% RSLogix 500 project PV5.RSS, saved by version 8.30.00.16 %
PROJECT "PV5"    % processor: Bul.1763 MicroLogix 1100 Series B %

PROGRAM FILES
  LAD 2   25 rungs

DATA FILES
  O0 OUTPUT  5 elements
  I1 INPUT  7 elements
  S2 STATUS  66 elements
  B3 BINARY  2 elements
  T4 TIMER  3 elements
  C5 COUNTER  1 elements
  R6 CONTROL  1 elements
  N7 INTEGER  3 elements
  F8 FLOAT  1 elements

LADDER 2
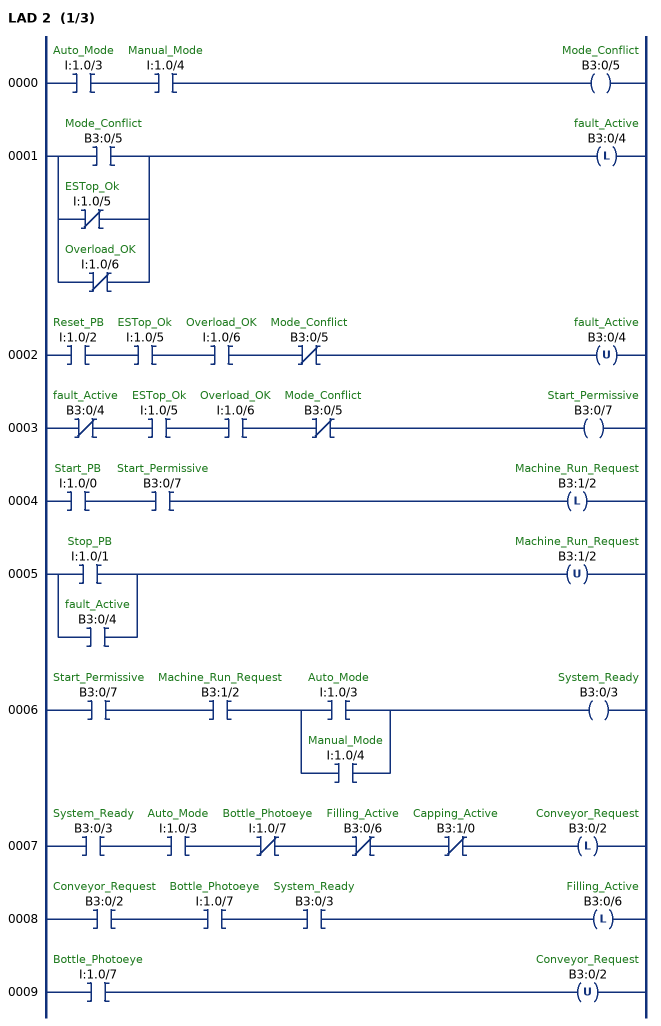
% Rung: 0 %
SOR XIC I:1.0/3 XIC I:1.0/4 OTE B3:0/5 EOR
%   I:1.0/3  "Auto_Mode" %
%   I:1.0/4  "Manual_Mode" %
%   B3:0/5  "Mode_Conflict" %
% Rung: 1 %
SOR BST XIC B3:0/5 NXB BST XIO I:1.0/5 NXB XIO I:1.0/6 BND BND OTL B3:0/4 EOR
%   B3:0/5  "Mode_Conflict" %
%   I:1.0/5  "ESTop_Ok" %
%   I:1.0/6  "Overload_OK" %
%   B3:0/4  "fault_Active" %
% Rung: 2 %
SOR XIC I:1.0/2 XIC I:1.0/5 XIC I:1.0/6 XIO B3:0/5 OTU B3:0/4 EOR
%   I:1.0/2  "Reset_PB" %
%   I:1.0/5  "ESTop_Ok" %
%   I:1.0/6  "Overload_OK" %
%   B3:0/5  "Mode_Conflict" %
%   B3:0/4  "fault_Active" %
% Rung: 3 %
SOR XIO B3:0/4 XIC I:1.0/5 XIC I:1.0/6 XIO B3:0/5 OTE B3:0/7 EOR
%   B3:0/4  "fault_Active" %
%   I:1.0/5  "ESTop_Ok" %
%   I:1.0/6  "Overload_OK" %
%   B3:0/5  "Mode_Conflict" %
%   B3:0/7  "Start_Permissive" %
% Rung: 4 %
SOR XIC I:1.0/0 XIC B3:0/7 OTL B3:1/2 EOR
%   I:1.0/0  "Start_PB" %
%   B3:0/7  "Start_Permissive" %
%   B3:1/2  "Machine_Run_Request" %
% Rung: 5 %
SOR BST XIC I:1.0/1 NXB XIC B3:0/4 BND OTU B3:1/2 EOR
%   I:1.0/1  "Stop_PB" %
%   B3:0/4  "fault_Active" %
%   B3:1/2  "Machine_Run_Request" %
% Rung: 6 %
SOR XIC B3:0/7 XIC B3:1/2 BST XIC I:1.0/3 NXB XIC I:1.0/4 BND OTE B3:0/3 EOR
%   B3:0/7  "Start_Permissive" %
%   B3:1/2  "Machine_Run_Request" %
%   I:1.0/3  "Auto_Mode" %
%   I:1.0/4  "Manual_Mode" %
%   B3:0/3  "System_Ready" %
% Rung: 7 %
SOR XIC B3:0/3 XIC I:1.0/3 XIO I:1.0/7 XIO B3:0/6 XIO B3:1/0 OTL B3:0/2 EOR
%   B3:0/3  "System_Ready" %
%   I:1.0/3  "Auto_Mode" %
%   I:1.0/7  "Bottle_Photoeye" %
%   B3:0/6  "Filling_Active" %
%   B3:1/0  "Capping_Active" %
%   B3:0/2  "Conveyor_Request" %
% Rung: 8 %
SOR XIC B3:0/2 XIC I:1.0/7 XIC B3:0/3 OTL B3:0/6 EOR
%   B3:0/2  "Conveyor_Request" %
%   I:1.0/7  "Bottle_Photoeye" %
%   B3:0/3  "System_Ready" %
%   B3:0/6  "Filling_Active" %
% Rung: 9 %
SOR XIC I:1.0/7 OTU B3:0/2 EOR
%   I:1.0/7  "Bottle_Photoeye" %
%   B3:0/2  "Conveyor_Request" %

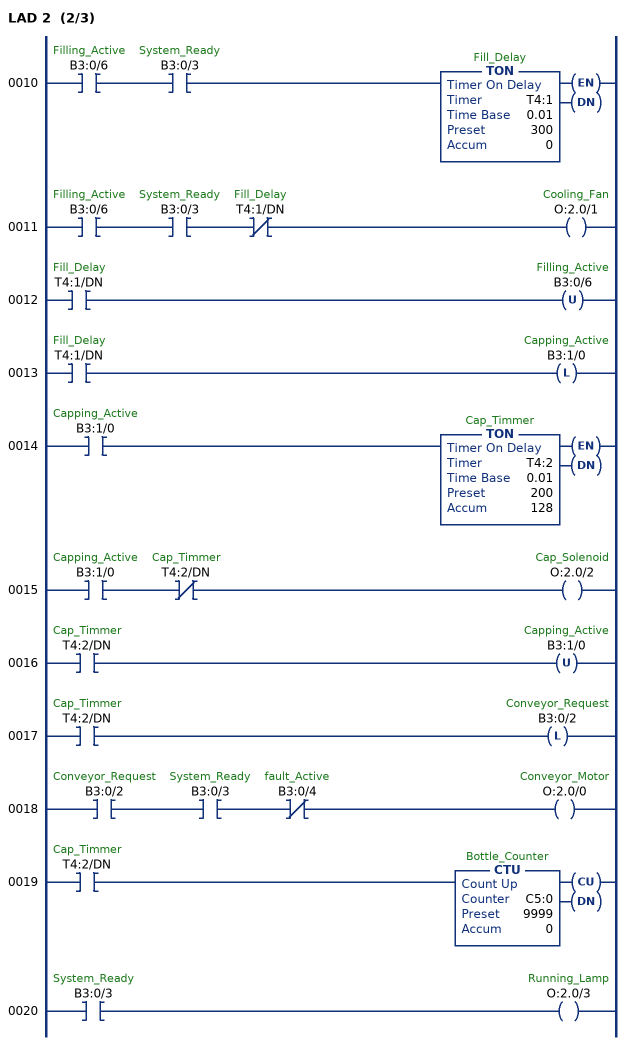
% Rung: 10 %
SOR XIC B3:0/6 XIC B3:0/3 TON T4:1 0.01 300 0 EOR
%   B3:0/6  "Filling_Active" %
%   B3:0/3  "System_Ready" %
%   T4:1  "Fill_Delay" %
% Rung: 11 %
SOR XIC B3:0/6 XIC B3:0/3 XIO T4:1/DN OTE O:2.0/1 EOR
%   B3:0/6  "Filling_Active" %
%   B3:0/3  "System_Ready" %
%   T4:1  "Fill_Delay" %
%   O:2.0/1  "Cooling_Fan" %
% Rung: 12 %
SOR XIC T4:1/DN OTU B3:0/6 EOR
%   T4:1  "Fill_Delay" %
%   B3:0/6  "Filling_Active" %
% Rung: 13 %
SOR XIC T4:1/DN OTL B3:1/0 EOR
%   T4:1  "Fill_Delay" %
%   B3:1/0  "Capping_Active" %
% Rung: 14 %
SOR XIC B3:1/0 TON T4:2 0.01 200 128 EOR
%   B3:1/0  "Capping_Active" %
%   T4:2  "Cap_Timmer" %
% Rung: 15 %
SOR XIC B3:1/0 XIO T4:2/DN OTE O:2.0/2 EOR
%   B3:1/0  "Capping_Active" %
%   T4:2  "Cap_Timmer" %
%   O:2.0/2  "Cap_Solenoid" %
% Rung: 16 %
SOR XIC T4:2/DN OTU B3:1/0 EOR
%   T4:2  "Cap_Timmer" %
%   B3:1/0  "Capping_Active" %
% Rung: 17 %
SOR XIC T4:2/DN OTL B3:0/2 EOR
%   T4:2  "Cap_Timmer" %
%   B3:0/2  "Conveyor_Request" %
% Rung: 18 %
SOR XIC B3:0/2 XIC B3:0/3 XIO B3:0/4 OTE O:2.0/0 EOR
%   B3:0/2  "Conveyor_Request" %
%   B3:0/3  "System_Ready" %
%   B3:0/4  "fault_Active" %
%   O:2.0/0  "Conveyor_Motor" %
% Rung: 19 %
SOR XIC T4:2/DN CTU C5:0 9999 0 EOR
%   T4:2  "Cap_Timmer" %
%   C5:0  "Bottle_Counter" %
% Rung: 20 %
SOR XIC B3:0/3 OTE O:2.0/3 EOR
%   B3:0/3  "System_Ready" %
%   O:2.0/3  "Running_Lamp" %

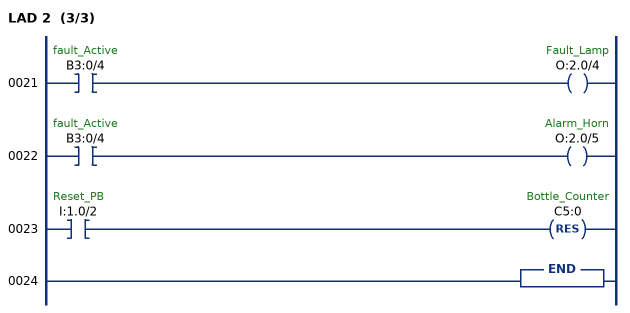
% Rung: 21 %
SOR XIC B3:0/4 OTE O:2.0/4 EOR
%   B3:0/4  "fault_Active" %
%   O:2.0/4  "Fault_Lamp" %
% Rung: 22 %
SOR XIC B3:0/4 OTE O:2.0/5 EOR
%   B3:0/4  "fault_Active" %
%   O:2.0/5  "Alarm_Horn" %
% Rung: 23 %
SOR XIC I:1.0/2 RES C5:0 EOR
%   I:1.0/2  "Reset_PB" %
%   C5:0  "Bottle_Counter" %
% Rung: 24 %
SOR END EOR

OTHER DOCUMENTED ADDRESSES
  B3:0/0  "Auto_Heating_Request"
  B3:0/1  "Manual_Run_Request"
  I:1.0/8  "High_Level_Switch"
  I:3.0/0  "High_Level_Switch"
  T4:0  "Delay_Timer"

DATA TABLE (non-zero values as saved)
DATA B3
% B3:0 % 0X0088 0X0005
DATA T4
% .PRE .ACC %
% T4:0 % 300 0
% T4:1 % 300 0
% T4:2 % 200 128
DATA C5
% .PRE .ACC %
% C5:0 % 9999 0
DATA N7
% N7:0 % 70 70 75
